SYSTEM TruckCaseStudy
  (* Version 1.0, 2022-12-15, AK124017 *)
  APPLICATION TruckCaseStudyApp
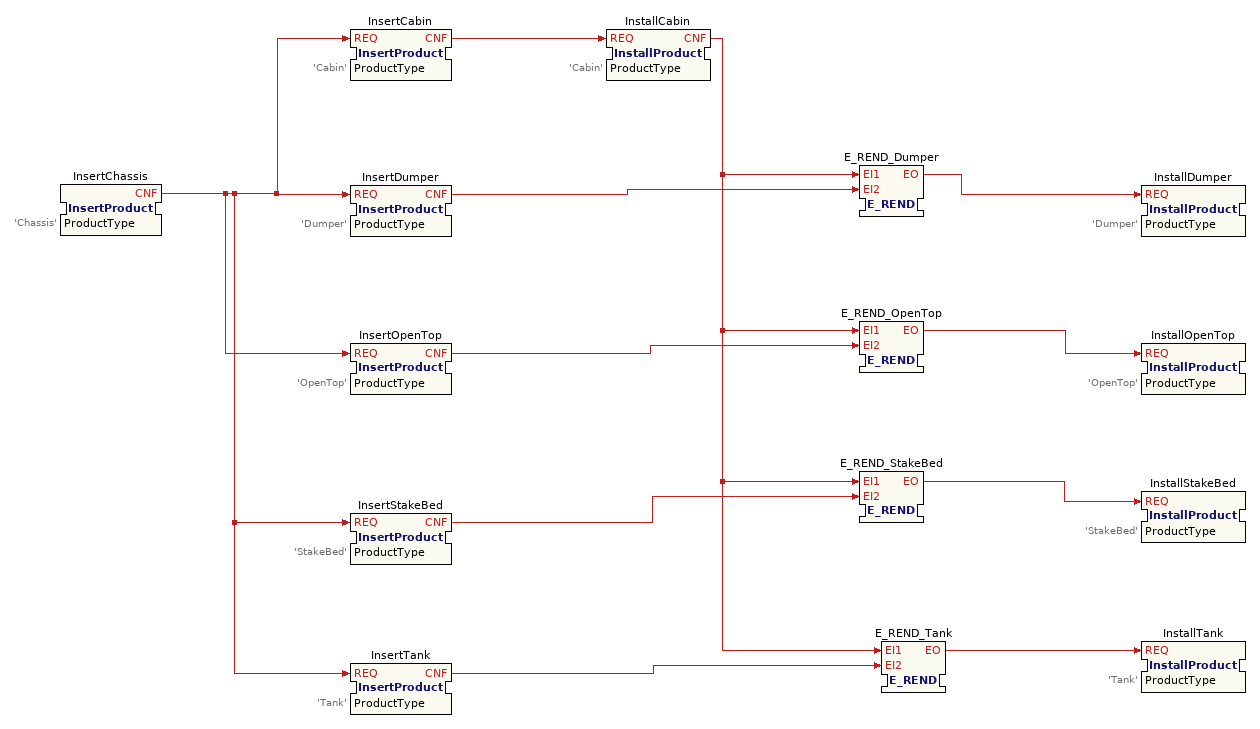
    FBS
      InsertChassis : InsertProduct(ProductType := 'Chassis');
      InsertCabin : InsertProduct(ProductType := 'Cabin');
      InstallOpenTop : InstallProduct(ProductType := 'OpenTop');
      InsertOpenTop : InsertProduct(ProductType := 'OpenTop');
      InstallCabin : InstallProduct(ProductType := 'Cabin');
      InsertDumper : InsertProduct(ProductType := 'Dumper');
      InstallDumper : InstallProduct(ProductType := 'Dumper');
      InsertStakeBed : InsertProduct(ProductType := 'StakeBed');
      InstallStakeBed : InstallProduct(ProductType := 'StakeBed');
      InsertTank : InsertProduct(ProductType := 'Tank');
      InstallTank : InstallProduct(ProductType := 'Tank');
      E_REND_Dumper : E_REND;
      E_REND_OpenTop : E_REND;
      E_REND_StakeBed : E_REND;
      E_REND_Tank : E_REND;
    END_FBS
    EVENT_CONNECTIONS
      InsertChassis.CNF TO InsertCabin.REQ;
      InsertChassis.CNF TO InsertOpenTop.REQ;
      InsertChassis.CNF TO InsertDumper.REQ;
      InsertCabin.CNF TO InstallCabin.REQ;
      InsertChassis.CNF TO InsertStakeBed.REQ;
      InsertChassis.CNF TO InsertTank.REQ;
      E_REND_Dumper.EO TO InstallDumper.REQ;
      InstallCabin.CNF TO E_REND_Dumper.EI1;
      InsertDumper.CNF TO E_REND_Dumper.EI2;
      InstallCabin.CNF TO E_REND_OpenTop.EI1;
      InstallCabin.CNF TO E_REND_StakeBed.EI1;
      InstallCabin.CNF TO E_REND_Tank.EI1;
      E_REND_OpenTop.EO TO InstallOpenTop.REQ;
      E_REND_StakeBed.EO TO InstallStakeBed.REQ;
      E_REND_Tank.EO TO InstallTank.REQ;
      InsertOpenTop.CNF TO E_REND_OpenTop.EI2;
      InsertStakeBed.CNF TO E_REND_StakeBed.EI2;
      InsertTank.CNF TO E_REND_Tank.EI2;
    END_CONNECTIONS
  END_APPLICATION
END_SYSTEM
